FUNCTION ReactivePower : Real
VAR_INPUT
	AppPower	: REAL;
	RealPower 	: REAL;
	PowerFactor	: REAL;
END_VAR
VAR
END_VAR

IF RealPower > AppPower THEN // NAN solution
	RETURN;
END_IF

IF powerfactor < 0 THEN
	ReactivePower := - SQRT(EXPT(AppPower, 2) - EXPT(RealPower,2));
ELSE
	ReactivePower := SQRT(EXPT(AppPower, 2) - EXPT(RealPower,2));
END_IF

END_FUNCTION

(* stored: Version 1.1.0.1, ProductVersion 3.1.4026.18
   POU ReactivePower: Id {f4ec3add-8d4b-421c-bd8a-a79afa8a4014}, SpecialFunc None *)
